PROGRAM PRG_MAIN
VAR

	test: BOOL;
	debug: INT;

END_VAR

//Recipes
Clock();


IF Config.Initialised() THEN   
	debug := debug+1;
	PRG_IO();
	PRG_Machine();
END_IF

END_PROGRAM

(* stored: Version 1.1.0.1, ProductVersion 3.1.4020.12
   POU PRG_MAIN: Id {d04c0ba0-8ee8-4b1d-b9a8-6a748878b094}, SpecialFunc None *)
